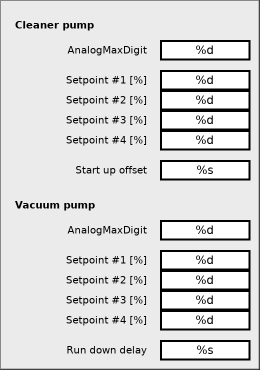
VISUALIZATION _VISU_CleanSequence  // 260x370
    Rectangle (0,0 260x370)
    Rectangle (160,40 90x20), "%d", text variable: PRG_MACHINE.fb_CleaningControl[PRG_MACHINE.iL_Sel_Module].fb_CleaningValvePump.lR_AnalogMaxDigitCleanerPump
        OnMouseDown: write the text variable via Default
    Rectangle (10,40 140x20), "AnalogMaxDigit"
    Rectangle (12,15 131x20), "Cleaner pump"
    Rectangle (160,70 90x20), "%d", text variable: PRG_MACHINE.fb_CleaningControl[PRG_MACHINE.iL_Sel_Module].fb_CleaningValvePump.lR_SetPoint1CleanerPump
        OnMouseDown: write the text variable via Default, min 0, max 100
    Rectangle (10,70 140x20), "Setpoint #1 [%]"
    Rectangle (160,90 90x20), "%d", text variable: PRG_MACHINE.fb_CleaningControl[PRG_MACHINE.iL_Sel_Module].fb_CleaningValvePump.lR_SetPoint2CleanerPump
        OnMouseDown: write the text variable via Default, min 0, max 100
    Rectangle (10,90 140x20), "Setpoint #2 [%]"
    Rectangle (160,110 90x20), "%d", text variable: PRG_MACHINE.fb_CleaningControl[PRG_MACHINE.iL_Sel_Module].fb_CleaningValvePump.lR_SetPoint3CleanerPump
        OnMouseDown: write the text variable via Default, min 0, max 100
    Rectangle (10,110 140x20), "Setpoint #3 [%]"
    Rectangle (160,130 90x20), "%d", text variable: PRG_MACHINE.fb_CleaningControl[PRG_MACHINE.iL_Sel_Module].fb_CleaningValvePump.lR_SetPoint4CleanerPump
        OnMouseDown: write the text variable via Default, min 0, max 100
    Rectangle (10,130 140x20), "Setpoint #4 [%]"
    Rectangle (160,220 90x20), "%d", text variable: PRG_MACHINE.fb_CleaningControl[PRG_MACHINE.iL_Sel_Module].fb_CleaningValvePump.lR_AnalogMaxDigitVacuumPump
        OnMouseDown: write the text variable via Default
    Rectangle (10,220 140x20), "AnalogMaxDigit"
    Rectangle (12,195 131x20), "Vacuum pump"
    Rectangle (160,250 90x20), "%d", text variable: PRG_MACHINE.fb_CleaningControl[PRG_MACHINE.iL_Sel_Module].fb_CleaningValvePump.lR_SetPoint1VacuumPump
        OnMouseDown: write the text variable via Default, min 0, max 100
    Rectangle (10,250 140x20), "Setpoint #1 [%]"
    Rectangle (160,270 90x20), "%d", text variable: PRG_MACHINE.fb_CleaningControl[PRG_MACHINE.iL_Sel_Module].fb_CleaningValvePump.lR_SetPoint2VacuumPump
        OnMouseDown: write the text variable via Default, min 0, max 100
    Rectangle (10,270 140x20), "Setpoint #2 [%]"
    Rectangle (160,290 90x20), "%d", text variable: PRG_MACHINE.fb_CleaningControl[PRG_MACHINE.iL_Sel_Module].fb_CleaningValvePump.lR_SetPoint3VacuumPump
        OnMouseDown: write the text variable via Default, min 0, max 100
    Rectangle (10,290 140x20), "Setpoint #3 [%]"
    Rectangle (160,310 90x20), "%d", text variable: PRG_MACHINE.fb_CleaningControl[PRG_MACHINE.iL_Sel_Module].fb_CleaningValvePump.lR_SetPoint4VacuumPump
        OnMouseDown: write the text variable via Default, min 0, max 100
    Rectangle (10,310 140x20), "Setpoint #4 [%]"
    Rectangle (160,160 90x20), "%s", text variable: PRG_MACHINE.fb_CleaningControl[PRG_MACHINE.iL_Sel_Module].fb_CleaningValvePump.tR_CleanerPumpOffset
        OnMouseDown: write the text variable via Default
    Rectangle (10,160 140x20), "Start up offset"
    Rectangle (160,340 90x20), "%s", text variable: PRG_MACHINE.fb_CleaningControl[PRG_MACHINE.iL_Sel_Module].fb_CleaningValvePump.tR_VacuumPumpDelay
        OnMouseDown: write the text variable via Default
    Rectangle (10,340 140x20), "Run down delay"
END_VISUALIZATION

(* stored: Version 1.1.0.1, ProductVersion 3.1.4024.11
   Visu _VISU_CleanSequence: Id {394e0fd8-0f39-4b98-88d4-17226341e853} *)
